# EPICS substitutions: iocBoot/iocxxx/common/fb_epid.substitutions
# $Id$

file "$(OPTICS)/opticsApp/Db/fb_epid.db"
  {
    {
        P="$(PREFIX)epid1",
	IN="$(PREFIX)epid1:sim.VAL",
	OUT="$(PREFIX)epid1:sim.D",
	MODE=PID,
	CALC=A,
	PERMIT1="$(PREFIX)epid1:on.VAL",
	PERMIT2="",
	PERMIT3="",
	PERMIT4=""
    }
  }
